// SIMATIC S7-200 project (STEP 7-Micro/WIN), CPU 226 CN REL 02.01

ORGANIZATION_BLOCK 主程序:OB1
TITLE=程序注释
BEGIN
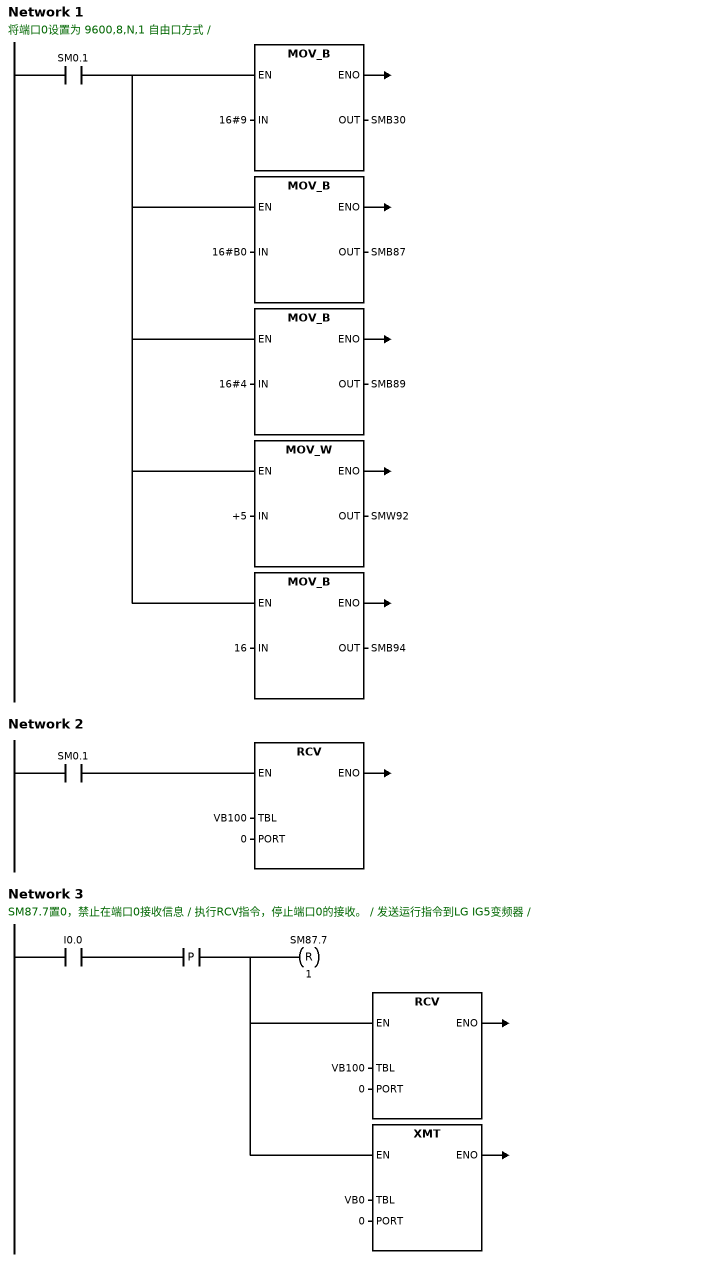
Network 1
// 将端口0设置为 9600,8,N,1 自由口方式
// 
LD     SM0.1
MOVB   16#9, SMB30
MOVB   16#B0, SMB87
MOVB   16#4, SMB89
MOVW   +5, SMW92
MOVB   16, SMB94
Network 2
LD     SM0.1
RCV    VB100, 0
Network 3
// SM87.7置0，禁止在端口0接收信息
// 执行RCV指令，停止端口0的接收。
// 发送运行指令到LG IG5变频器
// 
LD     I0.0
EU
R      SM87.7, 1
RCV    VB100, 0
XMT    VB0, 0
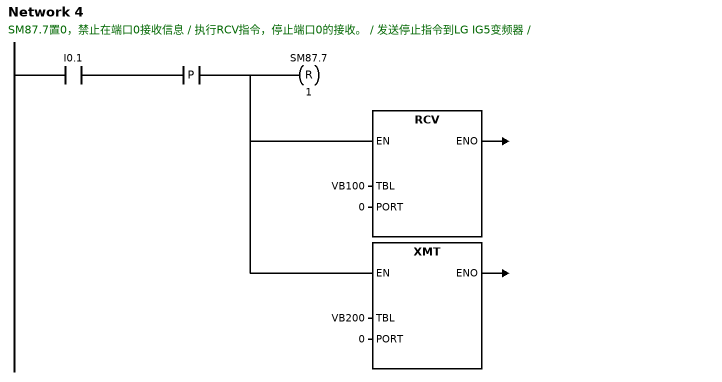
Network 4
// SM87.7置0，禁止在端口0接收信息
// 执行RCV指令，停止端口0的接收。
// 发送停止指令到LG IG5变频器
// 
LD     I0.1
EU
R      SM87.7, 1
RCV    VB100, 0
XMT    VB200, 0
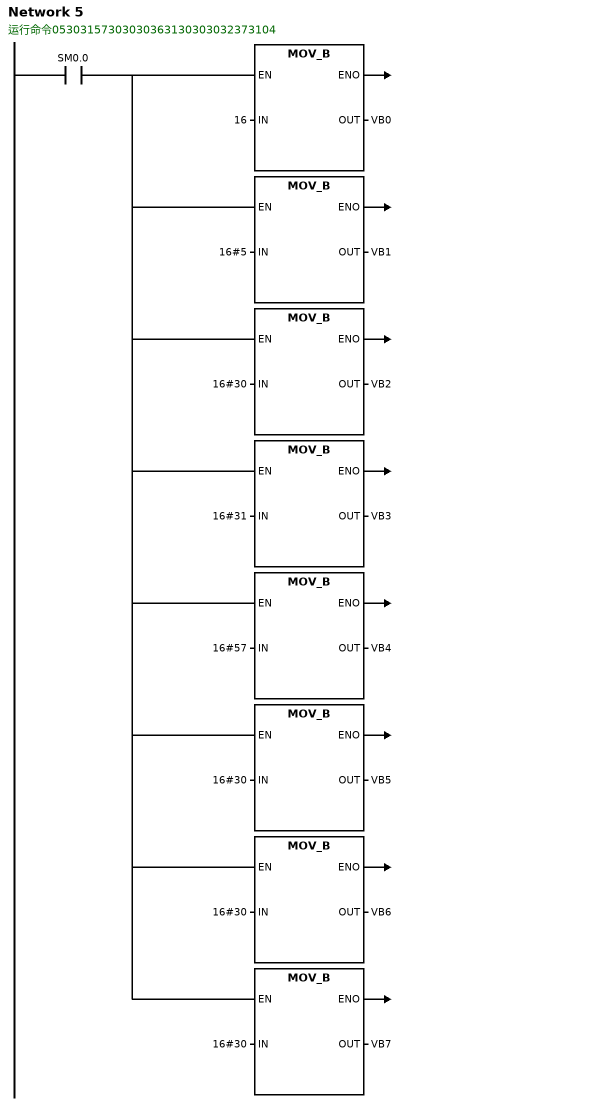
Network 5
// 运行命令05303157303030363130303032373104
LD     SM0.0
MOVB   16, VB0
MOVB   16#5, VB1
MOVB   16#30, VB2
MOVB   16#31, VB3
MOVB   16#57, VB4
MOVB   16#30, VB5
MOVB   16#30, VB6
MOVB   16#30, VB7
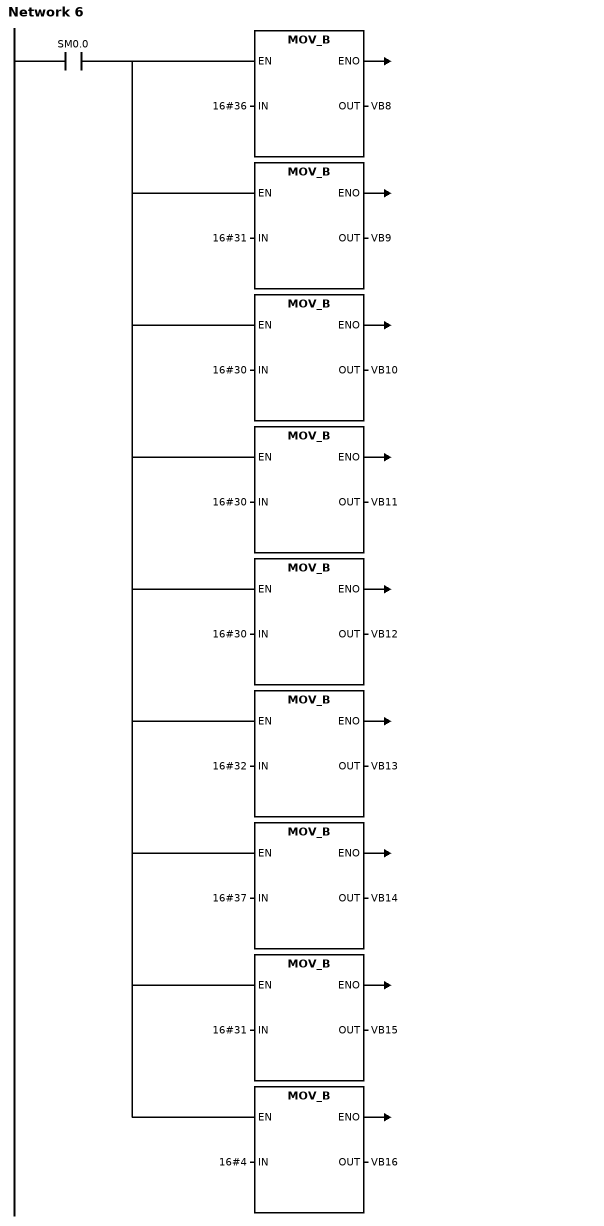
Network 6
LD     SM0.0
MOVB   16#36, VB8
MOVB   16#31, VB9
MOVB   16#30, VB10
MOVB   16#30, VB11
MOVB   16#30, VB12
MOVB   16#32, VB13
MOVB   16#37, VB14
MOVB   16#31, VB15
MOVB   16#4, VB16
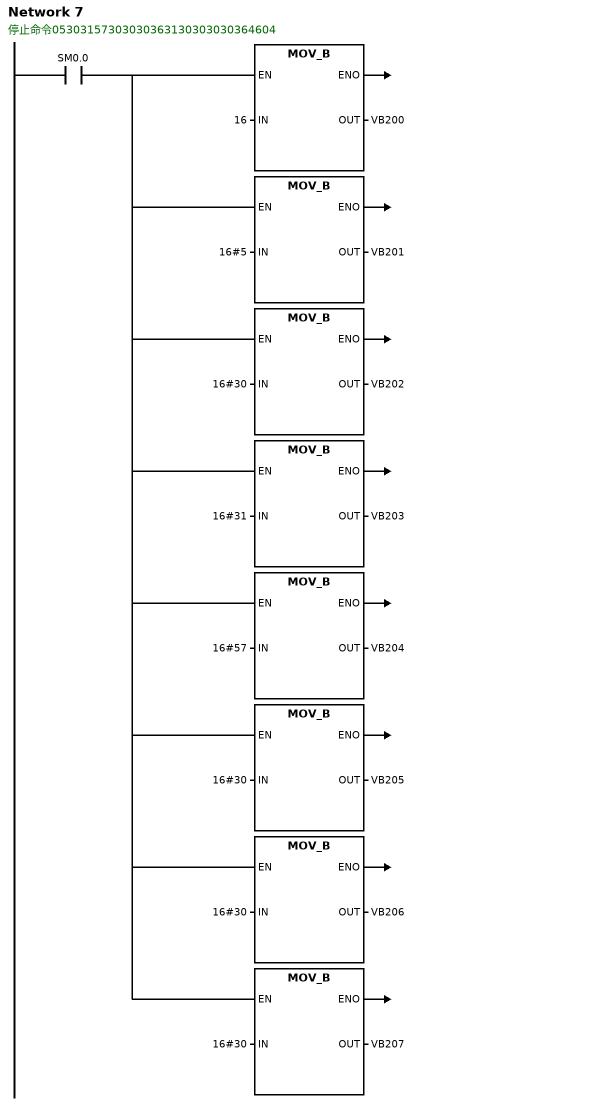
Network 7
// 停止命令05303157303030363130303030364604
LD     SM0.0
MOVB   16, VB200
MOVB   16#5, VB201
MOVB   16#30, VB202
MOVB   16#31, VB203
MOVB   16#57, VB204
MOVB   16#30, VB205
MOVB   16#30, VB206
MOVB   16#30, VB207
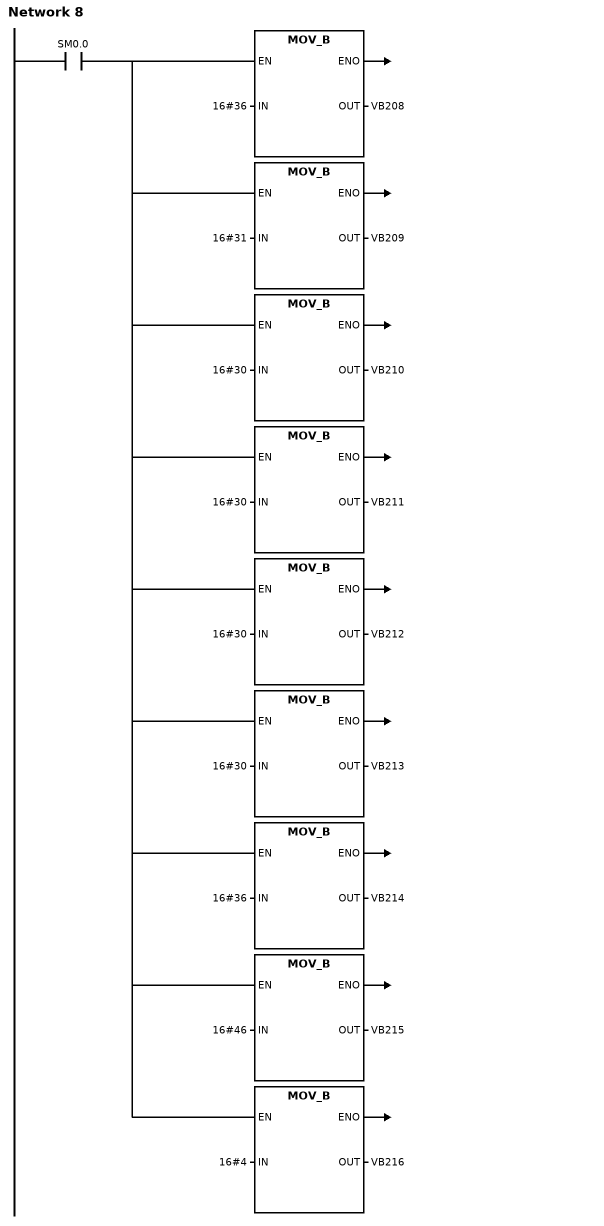
Network 8
LD     SM0.0
MOVB   16#36, VB208
MOVB   16#31, VB209
MOVB   16#30, VB210
MOVB   16#30, VB211
MOVB   16#30, VB212
MOVB   16#30, VB213
MOVB   16#36, VB214
MOVB   16#46, VB215
MOVB   16#4, VB216
END_ORGANIZATION_BLOCK
